FUNCTION F_SetOccupied : BOOL
(**************************************************************************************
 * 	Application		:	BoxControl Framework
 *	Revision		:	$Revision: 417092 $
 *	Revision date	:	$Date: 2018-11-14 12:58:58 +0100 (Mi., 14 Nov 2018) $
 *	Last changed by	:	$Author: q8aberh $
 *	URL				:	$URL: http://almscdc.swisslog.com/repo/SWPD/Development/ProMove/02_Controls/ProBox/03_Implementation/01_DevelopmentProject/01_Software/ProBox_COE/ProBox_DevProj_v1.0/PLC_1/20_Product/10_App/12_E_Functions/11_ProBox/02_Functions/F_SetOccupied.TcPOU $
 *
 *	Purpose			:	Return zone data
 *
 * ------------------------------------------------------------------------------------
 *	Copyright Swisslog [IP AG], Switzerland. All rights reserved.
 * 
 * ------------------------------------------------------------------------------------
 *	
 * 	Revision History: 
 *
 * 	VERSION			DATE			INITIALS			DESCRIPTION
 *	0.1				01.01.2001		swl					Example
 *
 **************************************************************************************)
VAR_INPUT
	eFunctionNumber		: E_FunctionNumber;
	ZoneNumber			: INT; 
END_VAR



// Check if function number and zone is valid
IF eFunctionNumber > E_FunctionNumber.F_BEGIN_FUNCTION AND
   eFunctionNumber < E_FunctionNumber.F_END_FUNCTION AND
   ZoneNumber > 0 AND ZoneNumber <= NUMBER_OF_ZONES_PER_FUNCTION THEN
  
	// Check reference is valid
    IF __ISVALIDREF(FunctionRegistry[eFunctionNumber].rFunction) THEN
	   // Return zone data
		IF __ISVALIDREF(FunctionRegistry[eFunctionNumber].Zone[ZoneNumber].refZoneData) THEN
			FunctionRegistry[eFunctionNumber].Zone[ZoneNumber].refZoneData.TransportControlData.Occupied := TRUE;
			FunctionRegistry[eFunctionNumber].Zone[ZoneNumber].refZoneData.TransportControlData.NumberOfPresentTUs :=1;
			FunctionRegistry[eFunctionNumber].Zone[ZoneNumber].refZoneData.TransportControlData.eTransportState := E_TransportState.OCCUPIED;
			F_SetOccupied:=TRUE;
	   END_IF
	    	   
    END_IF  
END_IF

END_FUNCTION

(* stored: Version 1.1.0.1, ProductVersion 3.1.4022.12
   POU F_SetOccupied: Id {b1673678-05b5-4936-a138-9e7fa8f823d8}, SpecialFunc None *)
